FUNCTION F_CheckAllStarted : BOOL
(**************************************************************************************
 * 	Application		:	BoxControl Framework
 *	Revision		:	$Revision: 417092 $
 *	Revision date	:	$Date: 2018-11-14 12:58:58 +0100 (Mi., 14 Nov 2018) $
 *	Last changed by	:	$Author: q8aberh $
 *	URL				:	$URL: http://almscdc.swisslog.com/repo/SWPD/Development/ProMove/02_Controls/ProBox/03_Implementation/01_DevelopmentProject/01_Software/ProBox_COE/ProBox_DevProj_v1.0/PLC_1/20_Product/10_App/12_E_Functions/11_ProBox/02_Functions/02_TransportControl/F_Che $
 *
 *	Purpose			:	Returns true if all the zones on the function are started
 *
 * ------------------------------------------------------------------------------------
 *	Copyright Swisslog [IP AG], Switzerland. All rights reserved.
 * 
 * ------------------------------------------------------------------------------------
 *	
 * 	Revision History: 
 *
 * 	VERSION			DATE			INITIALS			DESCRIPTION
 *	0.1				2018-08-14		PkF					First version
 *
 **************************************************************************************)
VAR_INPUT
	eFunctionNumber		: E_FunctionNumber; // Function number
END_VAR
VAR
	idx 				: INT; // Iterator
	AllStarted			: BOOL; // Temp to check if all zones are started
END_VAR

// Check if function number is valid
IF eFunctionNumber > E_FunctionNumber.F_BEGIN_FUNCTION AND
   eFunctionNumber < E_FunctionNumber.F_END_FUNCTION THEN
  
   // Check reference is valid
   IF __ISVALIDREF(FunctionRegistry[eFunctionNumber].rSettingsFunction) AND 
		__ISVALIDREF(FunctionRegistry[eFunctionNumber].rFunctionData) THEN
		// Return All Started
		AllStarted := TRUE;
		FOR idx := 1 TO FunctionRegistry[eFunctionNumber].rSettingsFunction.NumberOfZones DO
			IF (FunctionRegistry[eFunctionNumber].rFunctionData.OperationState.eState <> E_PositionState.STARTED AND 
				FunctionRegistry[eFunctionNumber].rFunctionData.OperationState.eState <> E_PositionState.STOPPING) OR 
				FunctionRegistry[eFunctionNumber].rFunctionData.ErrorData.ZoneErrorPending THEN
				AllStarted := FALSE;
				EXIT;
			END_IF
		END_FOR
		F_CheckAllStarted := AllStarted;
   END_IF
END_IF

END_FUNCTION

(* stored: Version 1.1.0.1, ProductVersion 3.1.4020.6
   POU F_CheckAllStarted: Id {ba29a7a0-b924-4ff3-849c-166fa6b8a7d3}, SpecialFunc None *)
